// TIA Portal V17 export
// export: Created 2024-09-02T12:50:21.9121913Z, ExportSetting WithDefaults, DisplayName Totally Integrated Automation Portal, DisplayVersion V17, DisplayName TIA Portal Openness, DisplayVersion V17, DisplayName TIA Portal Version Control Interface, DisplayVersion V17, DisplayName STEP 7 Professional, DisplayVersion V17, DisplayName STEP 7 Safety, DisplayVersion V17, DisplayName WinCC Professional, DisplayVersion V17
DATA_BLOCK "SysDI9_FG02_RF300_SLG2_OP70"   // DB1019
{ DB_Accessible_From_OPC_UA := 'FALSE' }
AUTHOR : STEAM
FAMILY : MOBY
NAME : MOBY
VERSION : 0.1
// stored: AutoNumber false, DBAccessibleFromOPCUA false, InstanceOfName SysFB_RF300, InstanceOfType FB
"SysFB_RF300"
   // VAR_INPUT
   //    HW_ID : Int;
   //    HW_ADR : Int;
   //    Channel : Int;
   //    RF_Type : Bool;
   //    "Fault ACK" : Bool;
   //    "New Start" : Bool;
   // END_VAR
   // VAR_OUTPUT
   //    Fault : Bool;
   //    "MDS Present" : Bool;
   //    HMIDiag : "TypeMobyHMIDiag";
   // END_VAR
   // VAR_IN_OUT
   //    Command : "TypeMobyBefehle";
   // END_VAR
   // VAR
   //    hwConnect { S7_SetPoint := 'True'} : IID_HW_CONNECT;
   //    Reset : Struct
   //       Start : Bool;
   //       Active : Bool;
   //       Finish : Bool;
   //       Fault : Bool;
   //       Status : DWord;
   //       Status_marked : DWord;
   //       Num_Of_OK : DInt;
   //       Num_Of_NOK : DInt;
   //       started : Bool;
   //       fp_started : Bool;
   //       hm_fp_started : Bool;
   //       Finish_OK : Bool;
   //       fp_Finish_OK : Bool;
   //       "hm fp_Finish_OK" : Bool;
   //       Finish_NOK : Bool;
   //       fp_Finish_NOK : Bool;
   //       "hm fp_Finish_NOK" : Bool;
   //       RunningTime : Time;
   //    END_STRUCT;
   //    Read : Struct
   //       Start : Bool;
   //       Active : Bool;
   //       Finish : Bool;
   //       Faul : Bool;
   //       MDS_present : Bool;
   //       Status : DWord;
   //       Status_marked : DWord;
   //       Num_Of_OK : DInt;
   //       Num_Of_NOK : DInt;
   //       started : Bool;
   //       fp_started : Bool;
   //       hm_fp_started : Bool;
   //       Finish_OK : Bool;
   //       fp_Finish_OK : Bool;
   //       "hm fp_Finish_OK" : Bool;
   //       Finish_NOK : Bool;
   //       fp_Finish_NOK : Bool;
   //       "hm fp_Finish_NOK" : Bool;
   //       RunningTime : Time;
   //    END_STRUCT;
   //    Write : Struct
   //       Start : Bool;
   //       Active : Bool;
   //       Finish : Bool;
   //       Fault : Bool;
   //       MDS_present : Bool;
   //       Status : DWord;
   //       Status_marked : DWord;
   //       Num_Of_OK : DInt;
   //       Num_Of_NOK : DInt;
   //       started : Bool;
   //       fp_started : Bool;
   //       hm_fp_started : Bool;
   //       Finish_OK : Bool;
   //       fp_Finish_OK : Bool;
   //       "hm fp_Finish_OK" : Bool;
   //       Finish_NOK : Bool;
   //       fp_Finish_NOK : Bool;
   //       "hm fp_Finish_NOK" : Bool;
   //       RunningTime : Time;
   //    END_STRUCT;
   //    SysDI_Reset { S7_SetPoint := 'True'} : Reset_RF300;
   //    SysDI_Read { S7_SetPoint := 'True'} : Read;
   //    SysDI_Write { S7_SetPoint := 'True'} : Write;
   //    SystemTime : Time;
   //    SystemTime_Old : Time;
   //    CycleTime : Time;
   //    ReadData : Struct
   //       SequenceNr : Int;
   //       RetVal : Word;
   //       Pos : DInt;
   //       finish : Bool;
   //    END_STRUCT;
   //    WriteData : Struct
   //       SequenceNr : Int;
   //       RetVal : Word;
   //       Pos : DInt;
   //       finish : Bool;
   //    END_STRUCT;
   //    ConnectionCheck : Struct
   //       TimeWithoutAction : Time;
   //       start : Bool;
   //       fp_start : Bool;
   //       HM_fp_start : Bool;
   //    END_STRUCT;
   //    "Checking Faults" : Struct
   //       FaultOccured : Bool;
   //       fp_FaultOccured : Bool;
   //       HM_fp_FaultOccured : Bool;
   //       TimeoutFault : Bool;
   //    END_STRUCT;
   //    SysDI_Reset200 { S7_SetPoint := 'True'} : Reset_RF200;
   // END_VAR
BEGIN
END_DATA_BLOCK
